# B&R Automation Studio project 2SegDemo (part 4)

#### Init.st - Init code
```iecst
PROGRAM _INIT
	ST_name(0,ADR(taskName),0);

	stationFbs.NCR_DemoFb.Controller := ADR(gMcAcp6DController);

	IF taskName = 'ProcSt1' THEN
		pStIf ACCESS ADR(gProcessStIf[STATION_1]);
		pStPars ACCESS ADR(gProcessRecipe.St1);

	ELSIF taskName = 'ProcSt2' THEN
		pStIf ACCESS ADR(gProcessStIf[STATION_2]);
		pStPars ACCESS ADR(gProcessRecipe.St2);
	END_IF

	gProcessStIf[STATION_1].Par.ShuttleIdx := STATION_IS_EMPTY;
	//Define station configuration values
	gProcessStIf[STATION_1].Cfg.StationPos.X := 0.66;
	gProcessStIf[STATION_1].Cfg.StationPos.Y := 0.54;

	gProcessStIf[STATION_2].Par.ShuttleIdx := STATION_IS_EMPTY;
	//Define station configuration values
	gProcessStIf[STATION_2].Cfg.StationPos.X := 0.30;
	gProcessStIf[STATION_2].Cfg.StationPos.Y := 0.66;

	gProcessRecipe.St1.OperationPos.X := 0.84;
	gProcessRecipe.St1.OperationPos.Y := 0.6;

	gProcessRecipe.St1.ExitPos.X := 0.66;
	gProcessRecipe.St1.ExitPos.Y := 0.66;

	gProcessRecipe.St2.OperationPos.X := 0.12;
	gProcessRecipe.St2.OperationPos.Y := 0.6;

	gProcessRecipe.St2.ExitPos.X := 0.30;
	gProcessRecipe.St2.ExitPos.Y := 0.54;
END_PROGRAM
```

#### Types.typ - Local data types
```iecst
TYPE
	StationStateEnum :
		(
		STATION_OFF, (*Station is currently disabled*)
		STATION_INIT, (*Station is initalizing*)
		STATION_WAIT_FOR_SHUTTLE, (*Station is waiting for a shuttle*)
		STATION_SH_ENTER,
		STATION_OPERATING, (*Station is preforming operation on shuttle*)
		STATION_SH_EXIT,
		STATION_DONE, (*Station is done with the process*)
		STATION_ERROR (*Station had an error*)
		);
	StationFbTyp : 	STRUCT
		Timer : TON;
		MovePlane : MC_BR_MoveInPlane_Acp6D;
		RunMacroFb : MC_BR_MacroRun_Acp6D;
		NCR_DemoFb : NonCenterRotationFb;
		MatrixFb : MatrixProcessFb;
	END_STRUCT;
	ProcessStationDemoEnum :
		(
		PROC_SPIRAL,
		PROC_MATRIX,
		PROC_Z_ROT,
		PROC_NCR
		);
END_TYPE
```

#### Variables.var - Local variables
```iecst
VAR
	state : StationStateEnum;
	stationFbs : StationFbTyp;
	stationPars : ProcessRecipeStationTyp;
	pStPars : REFERENCE TO ProcessRecipeStationTyp;
	pStIf : REFERENCE TO StationIfTyp;
	taskName : STRING[80];
	processDemoTyp : ProcessStationDemoEnum;
	matrixState : USINT;
END_VAR
```

#### LocalFunctions.fun
```iecst
{REDUND_ERROR} FUNCTION_BLOCK NonCenterRotationFb (* *) (*$GROUP=User,$CAT=User,$GROUPICON=User.png,$CATICON=User.png*)
	VAR_INPUT
		Execute : {REDUND_UNREPLICABLE} BOOL;
		Controller : REFERENCE TO McAcp6DControllerType;
		ShId : USINT;
	END_VAR
	VAR_OUTPUT
		Active : BOOL;
		DemoRunning : BOOL;
		Done : BOOL;
		Error : BOOL;
	END_VAR
	VAR
		Internal : NonCenterRotateInternalTyp;
	END_VAR
END_FUNCTION_BLOCK

FUNCTION_BLOCK MatrixProcessFb
	VAR_INPUT
		Execute : BOOL;
		Controller : REFERENCE TO McAcp6DControllerType;
		ShId : USINT;
		NumRows : UINT;
		NumColumns : UINT;
		RowSpacing : REAL; (*Spacing between rows in meters*)
		ColSpacing : REAL; (*Spacing between columns in meters*)
		Acceleration : REAL; (*Acceleration for movements m/s2*)
		Velocity : REAL; (*Velocity for movements in m/s*)
		FillTime : TIME; (*Time to wait at each fill station*)
	END_VAR
	VAR_OUTPUT
		Active : BOOL;
		CurrentPocket : UINT;
		Filling : BOOL;
		Done : BOOL;
		Error : BOOL;
	END_VAR
	VAR
		Internal : MatrixProcInternalTyp;
	END_VAR
END_FUNCTION_BLOCK
```

#### DemoFbsTypes.typ - Local data types
```iecst
(*Non Center Rotate Internal Typ*)

TYPE
	NonCenterRotateInternalTyp : 	STRUCT
		state : NCRStateEnum;
		errorState : NCRStateEnum;
		Fbs : NonCenterRotateFbsTyp;
	END_STRUCT;
	NCRStateEnum :
		(
		NCR_IDLE,
		NCR_MOVE_1,
		NCR_MOVE_2,
		NCR_MOVE_3,
		NCR_MOVE_4,
		NCR_MOVE_5,
		NCR_MOVE_6,
		NCR_DONE,
		NCR_ERROR,
		NCR_RESET
		);
	NonCenterRotateFbsTyp : 	STRUCT
		DelayTimerFb : TON;
		ShortAxisFb : MC_BR_MoveShortAxis_Acp6D;
		ShStopFb : MC_BR_Stop_Acp6D;
	END_STRUCT;
END_TYPE

(*Matrix Process Types*)

TYPE
	MatrixProcInternalTyp : 	STRUCT
		state : MatrixProcStateEnum;
		errorState : MatrixProcStateEnum;
		cRow : UINT;
		cCol : UINT;
		fillDir : MatrixFillDirType;
		Fbs : MatrixProcFbsTyp;
	END_STRUCT;
	MatrixProcFbsTyp : 	STRUCT
		MoveInPlaneFb : MC_BR_MoveInPlane_Acp6D;
		FillTimerFb : TON;
	END_STRUCT;
	MatrixProcStateEnum :
		(
		MAT_IDLE,
		MAT_MOVE,
		MAT_FILL,
		MAT_MOVE_BACK,
		MAT_DONE,
		MAT_ERROR,
		MAT_RESET
		);
	MatrixFillDirType :
		(
		FILL_RIGHT,
		FILL_LEFT
		);
END_TYPE
```

#### NonCenterRotationFb.st
```iecst
(* Demo implementation to showcase non center rotation capabilities*)
(*
	Will rotate a shuttle around 2 points some amount. The center location points are hardcoded for the AtxWest/PackExpo 2021 Demo layout
	Send start macro command to # of shuttles defined by input
	Wait Input Time
		Increment group count
	Repeat until group count * shuttlesPerGroup >= TotalShuttleCount
	Stop
		Send all shuttles to default height
	Error
	Reset

*)
FUNCTION_BLOCK NonCenterRotationFb
	CASE Internal.state OF
		NCR_IDLE: //******************************************************************************** Idle Wait State
			IF Execute THEN
				Active := TRUE;
				DemoRunning := TRUE;

				Internal.Fbs.ShortAxisFb.Controller := ADR(Controller);
				Internal.Fbs.ShortAxisFb.ShuttleID := ShId;
				Internal.Fbs.ShortAxisFb.RotationType := mcACP6D_SHORT_AX_ROTATION_CENTER;
				Internal.Fbs.ShortAxisFb.RotationCenterX := 0;
				Internal.Fbs.ShortAxisFb.RotationCenterY := 0.6;
				Internal.Fbs.ShortAxisFb.PositionZ := 0.00175;
				Internal.Fbs.ShortAxisFb.VelocityRz := 0.2;
				Internal.Fbs.ShortAxisFb.VelocityZ := 0.5;
				Internal.Fbs.ShortAxisFb.PositionRz := 0.080;
				Internal.state := NCR_MOVE_1;
			END_IF
		NCR_MOVE_1: //******************************************************************************** Move 1 state
			Internal.Fbs.ShortAxisFb.Execute := TRUE;

			IF Internal.Fbs.ShortAxisFb.Error THEN
				Error := TRUE;
				Internal.errorState := Internal.state;
				Internal.state := NCR_ERROR;
			ELSIF Internal.Fbs.ShortAxisFb.Acknowledge THEN
				Internal.Fbs.DelayTimerFb.PT := T#100ms;
				Internal.Fbs.DelayTimerFb.IN := TRUE;
				IF Internal.Fbs.DelayTimerFb.Q THEN
					Internal.Fbs.DelayTimerFb.IN := FALSE;
					Internal.Fbs.ShortAxisFb.Execute := FALSE;
					Internal.Fbs.ShortAxisFb.RotationCenterX := 0;
					Internal.Fbs.ShortAxisFb.RotationCenterY := 0.6;
					Internal.Fbs.ShortAxisFb.PositionRz := -0.080;

					Internal.state := NCR_MOVE_2;
				END_IF
			END_IF
		NCR_MOVE_2: //******************************************************************************** Move 2 state
			Internal.Fbs.ShortAxisFb.Execute := TRUE;

			IF Internal.Fbs.ShortAxisFb.Error THEN
				Error := TRUE;
				Internal.errorState := Internal.state;
				Internal.state := NCR_ERROR;
			ELSIF Internal.Fbs.ShortAxisFb.Acknowledge THEN
				Internal.Fbs.DelayTimerFb.PT := T#100ms;
				Internal.Fbs.DelayTimerFb.IN := TRUE;
				IF Internal.Fbs.DelayTimerFb.Q THEN
					Internal.Fbs.DelayTimerFb.IN := FALSE;
					Internal.Fbs.ShortAxisFb.Execute := FALSE;
					Internal.Fbs.ShortAxisFb.RotationCenterX := 0;
					Internal.Fbs.ShortAxisFb.RotationCenterY := 0.6;
					Internal.Fbs.ShortAxisFb.PositionRz := 0.0;

					Internal.state := NCR_MOVE_3;
				END_IF
			END_IF
		NCR_MOVE_3: //******************************************************************************** Move 3 state
			Internal.Fbs.ShortAxisFb.Execute := TRUE;

			IF Internal.Fbs.ShortAxisFb.Error THEN
				Error := TRUE;
				Internal.errorState := Internal.state;
				Internal.state := NCR_ERROR;
			ELSIF Internal.Fbs.ShortAxisFb.Acknowledge THEN
				Internal.Fbs.DelayTimerFb.PT := T#100ms;
				Internal.Fbs.DelayTimerFb.IN := TRUE;
				IF Internal.Fbs.DelayTimerFb.Q THEN
					Internal.Fbs.DelayTimerFb.IN := FALSE;
					Internal.Fbs.ShortAxisFb.Execute := FALSE;
					Internal.Fbs.ShortAxisFb.RotationCenterX := 0.9;
					Internal.Fbs.ShortAxisFb.RotationCenterY := 0.6;
					Internal.Fbs.ShortAxisFb.PositionRz := -0.08;

					Internal.state := NCR_MOVE_4;
				END_IF
			END_IF
		NCR_MOVE_4: //******************************************************************************** Move 4 state
			Internal.Fbs.ShortAxisFb.Execute := TRUE;

			IF Internal.Fbs.ShortAxisFb.Error THEN
				Error := TRUE;
				Internal.errorState := Internal.state;
				Internal.state := NCR_ERROR;
			ELSIF Internal.Fbs.ShortAxisFb.Acknowledge THEN
				Internal.Fbs.DelayTimerFb.PT := T#100ms;
				Internal.Fbs.DelayTimerFb.IN := TRUE;
				IF Internal.Fbs.DelayTimerFb.Q THEN
					Internal.Fbs.DelayTimerFb.IN := FALSE;
					Internal.Fbs.ShortAxisFb.Execute := FALSE;
					Internal.Fbs.ShortAxisFb.RotationCenterX := 0.9;
					Internal.Fbs.ShortAxisFb.RotationCenterY := 0.6;
					Internal.Fbs.ShortAxisFb.PositionRz := 0.080;

					Internal.state := NCR_MOVE_5;
				END_IF
			END_IF
		NCR_MOVE_5: //******************************************************************************** Move 5 state
			Internal.Fbs.ShortAxisFb.Execute := TRUE;

			IF Internal.Fbs.ShortAxisFb.Error THEN
				Error := TRUE;
				Internal.errorState := Internal.state;
				Internal.state := NCR_ERROR;
			ELSIF Internal.Fbs.ShortAxisFb.Acknowledge THEN
				Internal.Fbs.DelayTimerFb.PT := T#100ms;
				Internal.Fbs.DelayTimerFb.IN := TRUE;
				IF Internal.Fbs.DelayTimerFb.Q THEN
					Internal.Fbs.DelayTimerFb.IN := FALSE;
					Internal.Fbs.ShortAxisFb.Execute := FALSE;
					Internal.Fbs.ShortAxisFb.RotationCenterX := 0.9;
					Internal.Fbs.ShortAxisFb.RotationCenterY := 0.6;
					Internal.Fbs.ShortAxisFb.PositionRz := 0.0;

					Internal.state := NCR_MOVE_6;
				END_IF
			END_IF
		NCR_MOVE_6: //******************************************************************************** Move 6 state
			Internal.Fbs.ShortAxisFb.Execute := TRUE;

			IF Internal.Fbs.ShortAxisFb.Error THEN
				Error := TRUE;
				Internal.errorState := Internal.state;
				Internal.state := NCR_ERROR;
			ELSIF Internal.Fbs.ShortAxisFb.Done THEN //Wait for the last one to be done for the movement to be completely finished
				Internal.Fbs.DelayTimerFb.PT := T#100ms;
				Internal.Fbs.DelayTimerFb.IN := TRUE;
				IF Internal.Fbs.DelayTimerFb.Q THEN
					Internal.Fbs.DelayTimerFb.IN := FALSE;
					Internal.Fbs.ShortAxisFb.Execute := FALSE;

					Done := TRUE;

					Internal.state := NCR_DONE;
				END_IF
			END_IF
		NCR_DONE: //******************************************************************************** Done State
			IF NOT Execute THEN
				Internal.state := NCR_RESET;
			END_IF
		NCR_ERROR: //******************************************************************************** Error Present State
			IF NOT Execute THEN
				Internal.state := NCR_RESET;
			END_IF
		NCR_RESET: //******************************************************************************** Reset State

			Internal.Fbs.ShortAxisFb.Execute := FALSE;
			Internal.Fbs.ShStopFb.Execute := FALSE;
			Internal.Fbs.DelayTimerFb.IN := FALSE;

			Active := FALSE;
			DemoRunning := FALSE;
			Error := FALSE;
			Done := FALSE;

			Internal.state := NCR_IDLE;
	END_CASE;

	//Function block calls
	Internal.Fbs.DelayTimerFb();
	Internal.Fbs.ShStopFb();
	Internal.Fbs.ShortAxisFb();

END_FUNCTION_BLOCK
```

#### MatrixProcessFb.st
```iecst
(* implementation of a matrix movement process*)
(*
	Moves a shuttle in a matrix square pattern
	Assuming the following pattern, will move to the location -x,-y first
	  0 1 2
	2 x x x
	1 x x x
	0 o x x

	Will make a "snake" path through the matrix (move to the right, then to the left, repeat)

	Pauses at each location for the defined time

*)
FUNCTION_BLOCK MatrixProcessFb
	CASE Internal.state OF
		MAT_IDLE: //******************************************************************************** Idle Wait State
			IF Execute THEN
				Active := TRUE;

				Internal.cCol := 0;
				Internal.cRow := 0;
				CurrentPocket := 1;

				Internal.Fbs.MoveInPlaneFb.Controller := ADR(Controller);
				Internal.Fbs.MoveInPlaneFb.ShuttleID := ShId;
				Internal.Fbs.MoveInPlaneFb.Velocity := Velocity;
				Internal.Fbs.MoveInPlaneFb.Acceleration := Acceleration;
				Internal.Fbs.MoveInPlaneFb.Mode := mcACP6D_MOVE_RELATIVE;
				//This is a temporary fix for time constraints on the demo. This will only work for the 3x3 design in this demo
//				Internal.Fbs.MoveInPlaneFb.PositionX := - (ColSpacing * UINT_TO_REAL(NumColumns) / 2.0);
//				Internal.Fbs.MoveInPlaneFb.PositionY := - (RowSpacing * UINT_TO_REAL(NumRows) / 2.0);
				Internal.Fbs.MoveInPlaneFb.PositionX := - ColSpacing;
				Internal.Fbs.MoveInPlaneFb.PositionY := - RowSpacing;
				Internal.Fbs.MoveInPlaneFb.Execute := TRUE;

				Internal.state := MAT_MOVE;

			END_IF
		MAT_MOVE: //******************************************************************************** Moving State

			IF Internal.Fbs.MoveInPlaneFb.Error THEN
				Error := TRUE;
				Internal.errorState := Internal.state;
				Internal.state := MAT_ERROR;
			ELSIF Internal.Fbs.MoveInPlaneFb.Done THEN
				Internal.Fbs.MoveInPlaneFb.Execute := FALSE;

				Filling := TRUE;

				Internal.Fbs.FillTimerFb.PT := FillTime;
				Internal.Fbs.FillTimerFb.IN := TRUE;

				Internal.state := MAT_FILL;
			END_IF
		MAT_FILL: //******************************************************************************** Filling State
			IF Internal.Fbs.FillTimerFb.Q THEN
				Internal.Fbs.FillTimerFb.IN := FALSE;
				Filling := FALSE;

				IF Internal.fillDir = FILL_RIGHT THEN
					Internal.cCol := Internal.cCol + 1;
				ELSE
					Internal.cCol := Internal.cCol - 1;
				END_IF

				IF Internal.cCol >= NumColumns OR Internal.cCol <= 0 THEN
					//Finished a row
					Internal.cRow := Internal.cRow + 1;
					IF Internal.cRow >= NumRows THEN
						//Done
						Done := TRUE;

						Internal.state := MAT_DONE;
					ELSE
						IF Internal.fillDir = FILL_RIGHT THEN
							Internal.fillDir := FILL_LEFT;
							Internal.cCol := NumColumns;
						ELSE
							Internal.fillDir := FILL_RIGHT;
							Internal.cCol := 0;
						END_IF
						Internal.Fbs.MoveInPlaneFb.PositionX := 0;
						Internal.Fbs.MoveInPlaneFb.PositionY := RowSpacing;
						Internal.Fbs.MoveInPlaneFb.Execute := TRUE;
						CurrentPocket := CurrentPocket + 1;
						Internal.state := MAT_MOVE;
					END_IF
				ELSE
					IF Internal.fillDir = FILL_RIGHT THEN
						Internal.Fbs.MoveInPlaneFb.PositionX := ColSpacing;
					ELSE
						Internal.Fbs.MoveInPlaneFb.PositionX := -ColSpacing;
					END_IF
					Internal.Fbs.MoveInPlaneFb.PositionY := 0;
					Internal.Fbs.MoveInPlaneFb.Execute := TRUE;
					Internal.state := MAT_MOVE;
					CurrentPocket := CurrentPocket + 1;
				END_IF
			END_IF
		MAT_DONE: //******************************************************************************** Finished with the process
			IF NOT Execute THEN
				Internal.state := MAT_RESET;
			END_IF
		MAT_ERROR: //******************************************************************************** Error State
			IF NOT Execute THEN
				Internal.state := MAT_RESET;
			END_IF
		MAT_RESET: //******************************************************************************** Reset State
			Active := FALSE;
			Done := FALSE;
			Error := FALSE;
			CurrentPocket := 0;
			Filling := 0;

			Internal.cCol := 0;
			Internal.cRow := 0;
			Internal.fillDir := FILL_RIGHT;
			Internal.Fbs.FillTimerFb.IN := FALSE;
			Internal.Fbs.MoveInPlaneFb.Execute := FALSE;

			IF NOT Internal.Fbs.MoveInPlaneFb.Error THEN
				Internal.state := MAT_IDLE;
			END_IF
	END_CASE;

	//Function block calls
	Internal.Fbs.MoveInPlaneFb();
	Internal.Fbs.FillTimerFb();

END_FUNCTION_BLOCK
```

### Program Logical/Source/ProcessStations/InspectSt (IEC)

#### Types.typ
```iecst
TYPE
	InspectStationStateEnum :
		(
		INSPECT_OFF, (*Inspect station is currently disabled*)
		INSPECT_INIT, (*Inspect station is initalizing*)
		INSPECT_WAIT_FOR_SHUTTLE, (*Inspect Station is waiting for a shuttle*)
		INSPECT_INSPECTING, (*Inspect station is inspecting product on the shuttle*)
		INSPECT_WAIT_FOR_UNLOAD_ENABLE,
		INSPECT_DONE, (*Inspect station is done with the inspection process*)
		INSPECT_ERROR (*Inspect station had an error*)
		);
	InspectStationFbTyp : 	STRUCT
		Timer : TON;
		LedTimer : TOF;
	END_STRUCT;
END_TYPE
```

#### Variables.var
```iecst
VAR
	state : InspectStationStateEnum;
	stationFbs : InspectStationFbTyp;
	stationPars : ProcessRecipeStationTyp;
	LedTime : TIME;
END_VAR
```

#### Cyclic.st
```iecst
PROGRAM _CYCLIC

	IF NOT gInspectIf.Cmd.LocalOverride THEN
		stationPars := gProcessRecipe.Inspect;
	END_IF

	CASE state OF
		INSPECT_OFF: //********************************************************************************Load station is currently disabled
			IF gInspectIf.Cmd.Enable THEN
				state := INSPECT_INIT;
			ELSIF gInspectIf.Cmd.Reset THEN
				state := INSPECT_ERROR;
			END_IF
		INSPECT_INIT: //********************************************************************************Load station is initalizing
			gInspectIf.Sts.ReadyForNewShuttle := TRUE;
			gInspectIf.Sts.Enabled := TRUE;

			state := INSPECT_WAIT_FOR_SHUTTLE;
		INSPECT_WAIT_FOR_SHUTTLE: //********************************************************************************Load station is waiting for a shuttle to be present
			IF NOT gInspectIf.Cmd.Enable THEN
				gInspectIf.Sts.ReadyForNewShuttle := FALSE;
				gInspectIf.Sts.Enabled := FALSE;
				state := INSPECT_OFF;
			ELSIF gInspectIf.Par.ShuttleIdx <> STATION_IS_EMPTY AND gInspectIf.Cmd.Process THEN
				gInspectIf.Sts.ReadyForNewShuttle := FALSE;
				gInspectIf.Sts.Processing := TRUE;

				stationFbs.Timer.IN := TRUE;
				stationFbs.Timer.PT := stationPars.DwellTime;

				stationFbs.LedTimer.IN := TRUE;
				stationFbs.LedTimer.PT := LedTime;
				state := INSPECT_INSPECTING;
			END_IF
		INSPECT_INSPECTING:
			IF stationFbs.LedTimer.Q THEN
				stationFbs.LedTimer.IN := FALSE;
			END_IF
			IF stationFbs.Timer.Q THEN
				stationFbs.Timer.IN := FALSE;

				state := INSPECT_WAIT_FOR_UNLOAD_ENABLE;
			END_IF
		INSPECT_WAIT_FOR_UNLOAD_ENABLE:
			IF gUnloadStIf.Sts.Enabled THEN
				gInspectIf.Sts.Processing := FALSE;
				gInspectIf.Sts.Done := TRUE;
				gShuttleIf[gInspectIf.Par.ShuttleIdx].Cmd.NextStep := TRUE;

				state := INSPECT_DONE;
			ELSIF NOT gInspectIf.Cmd.Enable THEN
				gInspectIf.Sts.Done := FALSE;
				gInspectIf.Sts.Enabled := FALSE;
				gInspectIf.Sts.ReadyForNewShuttle := FALSE;
				gInspectIf.Sts.Processing := FALSE;
				stationFbs.Timer.IN := FALSE;

				gInspectIf.Par.ShuttleIdx := STATION_IS_EMPTY;
				state := INSPECT_OFF;
			END_IF
		INSPECT_DONE: //********************************************************************************Load station is done with the load process
			IF NOT gInspectIf.Cmd.Enable THEN
				gInspectIf.Sts.Done := FALSE;
				gInspectIf.Sts.Enabled := FALSE;
				gInspectIf.Sts.ReadyForNewShuttle := FALSE;
				stationFbs.Timer.IN := FALSE;
				gInspectIf.Sts.Processing := FALSE;

				gInspectIf.Par.ShuttleIdx := STATION_IS_EMPTY;
				state := INSPECT_OFF;
			ELSE
				gInspectIf.Cmd.Process := FALSE;
				gInspectIf.Par.ShuttleIdx := STATION_IS_EMPTY;
				gInspectIf.Sts.Done := FALSE;
				gInspectIf.Sts.ReadyForNewShuttle := TRUE;

				state := INSPECT_WAIT_FOR_SHUTTLE;
			END_IF

		INSPECT_ERROR: //********************************************************************************Load station had an error
			IF gInspectIf.Cmd.Reset THEN
				gInspectIf.Cmd.Reset := FALSE;

				gInspectIf.Sts.Done := FALSE;
				gInspectIf.Sts.Enabled := FALSE;
				gInspectIf.Sts.Error := FALSE;
				gInspectIf.Sts.Processing := FALSE;
				gInspectIf.Sts.ReadyForNewShuttle := FALSE;

				stationFbs.LedTimer.IN := FALSE;
				stationFbs.Timer.IN := FALSE;

				gInspectIf.Par.ShuttleIdx := STATION_IS_EMPTY;
				IF gInspectIf.Cmd.Enable THEN
					state := INSPECT_INIT;
				ELSE
					state := INSPECT_OFF;
				END_IF
			END_IF
	END_CASE;

	stationFbs.Timer();
	stationFbs.LedTimer();
END_PROGRAM
```

#### Init.st
```iecst
PROGRAM _INIT
	gInspectIf.Par.ShuttleIdx := STATION_IS_EMPTY;
	//Define station configuration values
	gInspectIf.Cfg.StationPos.X := 0.30;
	gInspectIf.Cfg.StationPos.Y := 0.30;
	LedTime := T#150ms;
END_PROGRAM
```

### Program Logical/Source/ProcessStations/CycChlCfg (IEC)

#### Types.typ
```iecst
TYPE
	CycChannelConfigStateEnum :
		(
		CFG_IDLE,
		CFG_CONFIG,
		CFG_ERROR
		);
	CycChannelCfgFbsTyp : 	STRUCT
		CfgReadCyclicPos : MC_BR_ConfigReadCyclicCh_Acp6D;
	END_STRUCT;
END_TYPE
```

#### Variables.var
```iecst
VAR
	state : CycChannelConfigStateEnum;
	Fbs : CycChannelCfgFbsTyp;
	logArgs : ARRAY[0..3] OF UDINT;
END_VAR
```

#### Cyclic.st
```iecst
PROGRAM _CYCLIC
	//Task that handles the configuration of the cyclic channels

	//Idle
	//Config
	//Error

	CASE state OF
		CFG_IDLE:  //********************************************************************************Idle state - wait for command
			IF gCyclicChlCfgIf.Cmds.Config THEN
				gCyclicChlCfgIf.Sts.Configuring := TRUE;
				gCyclicChlCfgIf.Sts.Ready := FALSE;

				Fbs.CfgReadCyclicPos.Controller := ADR(gMcAcp6DController);
				Fbs.CfgReadCyclicPos.NumberOfChannels := 2;

				Fbs.CfgReadCyclicPos.ChannelID[0] := 1;
				Fbs.CfgReadCyclicPos.ChannelID[1] := 2;
				Fbs.CfgReadCyclicPos.FeedbackMode[0] := mcACP6D_READ_CYCLIC_POSITION;
				Fbs.CfgReadCyclicPos.FeedbackMode[1] := mcACP6D_READ_CYCLIC_POSITION;

				//We must always configure 2 channels. In order to make it easier, channel 1 will always be the "load" channel and channel 2 will be the unload channel.
				//This means however that if there is no current shuttle in the station, we must still keep the channel enabled, so we're just going to use shuttle IDs 1 and 2 in the event
				//that there is no shuttle present
				IF gCyclicChlCfgIf.Pars.LoadShuttleIdx <> STATION_IS_EMPTY THEN
					Fbs.CfgReadCyclicPos.ShuttleID[0] := gShuttleIf[gCyclicChlCfgIf.Pars.LoadShuttleIdx].Cfg.ShuttleId;
				ELSE
					Fbs.CfgReadCyclicPos.ShuttleID[0] := 1;
				END_IF
				IF gCyclicChlCfgIf.Pars.UnloadShuttleIdx <> STATION_IS_EMPTY THEN
					Fbs.CfgReadCyclicPos.ShuttleID[1] := gShuttleIf[gCyclicChlCfgIf.Pars.UnloadShuttleIdx].Cfg.ShuttleId;
				ELSE
					Fbs.CfgReadCyclicPos.ShuttleID[1] := 2;
				END_IF
				Fbs.CfgReadCyclicPos.Execute := TRUE;

				state := CFG_CONFIG;
			END_IF

		CFG_CONFIG:  //********************************************************************************Configuration state - wait for status to report done/error
			IF Fbs.CfgReadCyclicPos.Error THEN
				logArgs[0] := ADR(Fbs.CfgReadCyclicPos.ShuttleID[0]);
				logArgs[1] := ADR(Fbs.CfgReadCyclicPos.ShuttleID[1]);
				logArgs[2] := ADR(Fbs.CfgReadCyclicPos.ErrorID);
				logFatal('CycChlCfg','Cyclic Channel configuration failed. Ch1 ID: %d CH2 ID: %d Error #: %d.',ADR(logArgs));
				state := CFG_ERROR;
			ELSIF Fbs.CfgReadCyclicPos.Done THEN
				gCyclicChlCfgIf.Cmds.Config := FALSE;
				gCyclicChlCfgIf.Sts.Configuring := FALSE;
				gCyclicChlCfgIf.Sts.Ready := TRUE;

				Fbs.CfgReadCyclicPos.Execute := FALSE;
				state := CFG_IDLE;
			END_IF
		CFG_ERROR:  //********************************************************************************Error State - wait for reset command
			Fbs.CfgReadCyclicPos.Execute := FALSE;

			//TODO: We'll need to reset the error flag (leaving it high just for debugging assistance)
			state := CFG_IDLE;

	END_CASE;
	//This is hard coded for 2 axes to get the X position cyclically for the two FBs

	 Fbs.CfgReadCyclicPos();
END_PROGRAM
```

#### Init.st
```iecst
PROGRAM _INIT
	gCyclicChlCfgIf.Sts.Ready := TRUE;

END_PROGRAM
```

- DoseHolder.blend (binary file, 866200 bytes)
- DoseHolder.blend1 (binary file, 866124 bytes)
- Visualisation Logical/mappView (not shown)

- DofRobot.gcode (not shown)

- RoutingRobotHelix.gcode (not shown)

- Test.gcode (not shown)

Listed in the project but not available here: Logical/Global.typ, Logical/Global.var, Logical/Source/ShuttleCtrl/ShCtrlGlobalVars.var, Logical/Source/ShuttleCtrl/ShCtrlGlobalTypes.typ, Logical/Source/Demos/VarDemos/Exit.st, Logical/Source/6DCtrl/Acp6DGlobalVars.var, Logical/Source/Auxil/AuxGlobalVars.var, Logical/Source/Auxil/AuxGlobalTypes.typ, Logical/Source/Auxil/AuditCtrl, Logical/Source/Auxil/OeeCalc, Logical/Source/ProcessStations/ProcessSt/Exit.st
